TYPE ST_BronkhorstMassFlowController_Options :
STRUCT
	fullyOpen	: BOOL;	// Opens controller fully
	fullyClose	: BOOL;	// Closes controller fully
END_STRUCT
END_TYPE

(* stored: Version 1.1.0.1, ProductVersion 3.1.4024.13
   DUT ST_BronkhorstMassFlowController_Options: Id {0d84a534-92a4-084b-39ed-aba80998cec7} *)
